FUNCTION_BLOCK FB_FT_PIWL (* Basic Function Block Type *)
  (* Standard: 61499-2; Classification: Control modules; Description: FT_PIWL is a PI controller with dynamic anti-wind Up. *)
  (* Version 0.0, 2011-08-25, 4DIAC-IDE, 4DIAC-Consortium *)
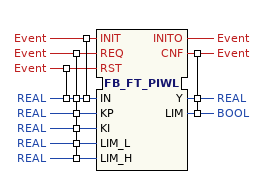
  EVENT_INPUT
    INIT WITH IN;
    REQ WITH IN, KP, KI, LIM_L, LIM_H; (* Normal Execution Request *)
    RST WITH IN;
  END_EVENT
  EVENT_OUTPUT
    INITO;
    CNF WITH Y, LIM; (* Execution Confirmation *)
  END_EVENT
  VAR_INPUT
    IN : REAL; (* input signal *)
    KP : REAL := 1.0; (* proportional gain of the controller *)
    KI : REAL := 1.0; (* integral gain of the controll *)
    LIM_L : REAL := -1.0E38; (* lower limit of the integrator output *)
    LIM_H : REAL := 1.0E38; (* upper limit of the integrator output *)
  END_VAR
  VAR_OUTPUT
    Y : REAL; (* output of the controller *)
    LIM : BOOL; (* TRUE if the output has reached a limit *)
  END_VAR
  VAR
    T_LAST : DWORD; (* Internal Variable *)
    IN_LAST : REAL; (* Internal Variable *)
    I : REAL; (* Internal Variable *)
    INIT : BOOL; (* Internal Variable *)
  END_VAR
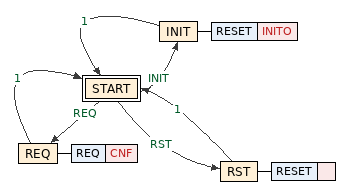
  EC_STATES
    START; (* Initial State *)
    INIT : RESET -> INITO; (* Initialization *)
    REQ : REQ -> CNF; (* Normal execution *)
    RST : RESET;
  END_STATES
  EC_TRANSITIONS
    START TO INIT := INIT;
    INIT TO START := 1;
    START TO REQ := REQ;
    REQ TO START := 1;
    START TO RST := RST;
    RST TO START := 1;
  END_TRANSITIONS
  ALGORITHM RESET IN ST: (* Initialization algorithm *)
INIT := true;
IN_LAST := IN;
T_LAST := T_PLC_US();
I := 0.0;
  END_ALGORITHM
  ALGORITHM REQ IN ST: (* Normally executed algorithm *)
(* TODO consider this in the export filter *)
VAR
	tx: DWORD;
	tc : REAL;
	p: REAL;
END_VAR


 (* read last cycle time in Microseconds *)
	tx := T_PLC_US();
	tc := DWORD_TO_REAL(tx - T_LAST);
	T_LAST := tx;

	(* calculate proportional part *)
	p := KP * IN;

	(* run integrator *)
	I := (IN + IN_LAST) * 5.0E-7 * KI * tc + I;
	IN_LAST := IN;

	(* calculate output Y *)
	Y := p + I;

	(* check output for limits *)
	IF Y >= LIM_H THEN
		Y := LIM_H;
		IF KI <> 0.0 THEN
			I := LIM_H - p;
		ELSE
			I := 0.0;
		END_IF;
		LIM := TRUE;
	ELSIF Y <= LIM_L THEN
		Y := LIM_L;
		IF KI <> 0.0 THEN
			I := LIM_L - p;
		ELSE
			I := 0.0;
		END_IF;
		LIM := TRUE;
	ELSE
		LIM := FALSE;
	END_IF;
  END_ALGORITHM
END_FUNCTION_BLOCK
